(* CoDeSys 2.3 export: WRITEVALUE.EXP *)

(* POU Functions/WriteValue, ST *)
FUNCTION WriteValue : BOOL
VAR_INPUT
	pValue : POINTER TO INT ; (**< Pointer to value to write *)
	Value : INT ; (**< Value to store into the variable *)
END_VAR
VAR
END_VAR
pValue ^ := Value;
END_FUNCTION
